// TIA Portal V17 export
// export: Created 2025-03-05T08:01:00.3212883Z, ExportSetting WithDefaults, DisplayName Totally Integrated Automation Portal, DisplayVersion V17 Update 8, DisplayName TIA Portal Openness, DisplayVersion V17 Update 8, DisplayName TIA Portal Version Control Interface, DisplayVersion V17, DisplayName SINAMICS Startdrive Advanced, DisplayVersion V17 SP2, DisplayName SINAMICS Startdrive G110M, G120, G120C, G120D, G120P, G115D, DisplayVersion V17 SP2, DisplayName SINAMICS Startdrive G130, G150, S120, S150, SINAMICS MV, S210, DisplayVersion V17 SP2, DisplayName STEP 7 Professional, DisplayVersion V17 Update 8, DisplayName SINUMERIK ONE STEP 7 Toolbox, DisplayVersion V17 Update 12, DisplayName SINUMERIK 840D sl STEP 7 Toolbox, DisplayVersion V17 Update 12, DisplayName STEP 7 Safety, DisplayVersion V17 Update 6, DisplayName WinCC Advanced, DisplayVersion V17 Update 8
DATA_BLOCK "LTLP_DirectKeyGetMovNoData"   // DB512
{ S7_Optimized_Access := 'FALSE'; DB_Accessible_From_OPC_UA := 'FALSE' }
VERSION : 0.1
// stored: AutoNumber false, DBAccessibleFromOPCUA false, DBAccessibleFromWebserver true, InstanceOfName LTLP_typeDirectKeyGetMoveNo, InstanceOfType UDT, IsOnlyStoredInLoadMemory false, IsWriteProtectedInAS false
"LTLP_typeDirectKeyGetMoveNo"
   // VAR
   //    PowerUp : Array[1..48] of Bool;
   //    Setup1 : Array[1..256] of Bool;
   //    Setup2 : Array[1..256] of Bool;
   //    PartMachining : Array[1..42] of Bool;
   //    CycleTypes : Array[1..16] of Bool;
   //    NutRunnerDeselection : Array[1..80] of Bool;
   //    GroupDeselection : Array[1..40] of Bool;
   //    Internal : Struct
   //       Last_PictureMask : Word;
   //       Last_SelIndex : Int;
   //    END_STRUCT;
   // END_VAR
BEGIN
END_DATA_BLOCK
